// TIA Portal project "P5_sim" (V14)
// Simulación planta envasadora de bolitas

(* hardware
DEVICE "S7-1200 station_1"  S7-1200 Station
   slot 0: "Rack_0"  S7-1200 Rack  Rack  V1.0
   slot 1: "PLC_1"  CPU 1214C DC/DC/DC  6ES7 214-1AG40-0XB0  V4.2
*)

// ===== PLC "PLC_1"  CPU 1214C DC/DC/DC =====

VAR_GLOBAL   // PLC tag table "Default tag table"
   ""I_PM"" AT %I0.0 : Bool;
   ""I_PP"" AT %I0.1 : Bool;
   ""Q_P2"" AT %Q0.1 : Bool;
   ""Q_P1"" AT %Q0.0 : Bool;
END_VAR